PROGRAM MAIN
VAR
	fbTimer: TP := (PT := TIME#3s0ms);
	bKnop AT %I*: BOOL := false;
	bLED1 AT %Q*: BOOL := FALSE;
END_VAR

fbTimer(IN:= bKnop, Q=>bLED1);

END_PROGRAM

(* stored: Version 1.1.0.1, ProductVersion 3.1.4024.12
   POU MAIN: Id {d2ddc2f6-b1b6-4f6a-8404-8d60b16ec7ea}, SpecialFunc None *)
